Universal Robots PolyScope program: base_b.urp

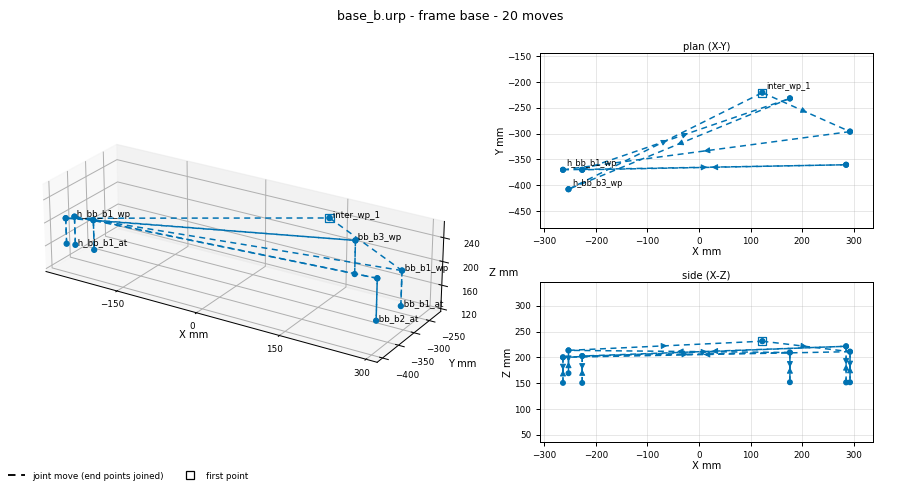
[picture p0: tool path of base_b.urp in frame base, 20 of 20 moves have a stored position in this frame; points joined in program order, loops and branches not executed]
Program base_b (installation=default directory=/programs/Session 1 createdIn=5.3.1.64192 lastSavedIn=5.3.1.64192 robotSerialNumber=20195300365)
Calibrated DH parameters: a=[-0.000093, -0.190649, -0.212673, 0.000091, -0.000205, 0]; d=[0.151591, 44.061648, -42.488068, -1.442789, 0.085322, 0.091911]; alpha=[1.570082, -0.003447, 0.007513, 1.572293, -1.571904, 0]; deltaTheta=[0, -0.672656, 0.728185, -0.055522, 0.000005, 0]
Robot Program (runOnlyOnce=true)
  URCap Gripper Activate (Robotiq_Grippers, Robotiq Inc.) dataModel(ResetAndActivateKey=false)
  URCap Gripper (Robotiq_Grippers, Robotiq Inc.) dataModel(position=50.0, force=100.0, speed=100.0, positionInDouble=50.0, forceInDouble=100.0, speedInDouble=100.0, slaveIds=[9], blocking=true)
  MoveJ speed 60 deg/s, acceleration 80 deg/s^2 (useActiveTCP=true) feature=Base
    Waypoint inter_wp_1: TCP in base x=122.78 y=-220.583 z=231.495 mm, rx=2.2968 ry=2.1205 rz=-0.0201 rad; joints [-29.631, -72.124, -124.848, -72.343, 89.412, -204.687] deg
  Folder Base_B
    MoveJ speed 60 deg/s, acceleration 80 deg/s^2 (useActiveTCP=true) feature=Base
      Waypoint bb_b1_wp: TCP in base x=292.658 y=-296.109 z=211.213 mm, rx=2.2199 ry=2.2113 rz=-0.0547 rad; joints [-26.688, -116.102, -82.488, -71.567, 88.238, -206.181] deg
      Waypoint bb_b1_at: TCP in base x=292.645 y=-296.127 z=151.887 mm, rx=2.2199 ry=2.2112 rz=-0.0548 rad; joints [-26.711, -122.1, -90.484, -57.573, 88.188, -206.122] deg
      URCap Gripper (Robotiq_Grippers, Robotiq Inc.) dataModel(position=100.0, force=100.0, speed=100.0, positionInDouble=100.0, forceInDouble=100.0, speedInDouble=100.0, slaveIds=[9], blocking=true)
      Waypoint bb_b1_wp: TCP in base x=292.658 y=-296.109 z=211.213 mm, rx=2.2199 ry=2.2113 rz=-0.0547 rad; joints [-26.688, -116.102, -82.488, -71.567, 88.238, -206.181] deg
      Waypoint h_bb_b1_wp: TCP in base x=-263.499 y=-370.068 z=200.329 mm, rx=-3.0828 ry=0.0524 rz=-0.0261 rad; joints [-108.781, -127.406, -65.833, -80.171, 90.182, -196.637] deg
      Waypoint h_bb_b1_at: TCP in base x=-263.484 y=-370.083 z=150.732 mm, rx=-3.0828 ry=0.0523 rz=-0.026 rad; joints [-108.797, -131.383, -72.897, -69.13, 90.158, -196.59] deg
      URCap Gripper (Robotiq_Grippers, Robotiq Inc.) dataModel(position=50.0, force=100.0, speed=100.0, positionInDouble=50.0, forceInDouble=100.0, speedInDouble=100.0, slaveIds=[9], blocking=true)
      Waypoint h_bb_b1_wp: TCP in base x=-263.499 y=-370.068 z=200.329 mm, rx=-3.0828 ry=0.0524 rz=-0.0261 rad; joints [-108.781, -127.406, -65.833, -80.171, 90.182, -196.637] deg
    MoveJ speed 60 deg/s, acceleration 80 deg/s^2 (useActiveTCP=true) feature=Base
      Waypoint bb_b2_wp: TCP in base x=285.029 y=-360.313 z=221.676 mm, rx=2.2402 ry=2.1488 rz=-0.0282 rad; joints [-34.898, -125.685, -65.053, -77.312, 88.836, -212.332] deg
      Waypoint bb_b2_at: TCP in base x=285.033 y=-360.322 z=151.608 mm, rx=2.2401 ry=2.1488 rz=-0.028 rad; joints [-34.925, -131.234, -75.256, -61.556, 88.801, -212.266] deg
      URCap Gripper (Robotiq_Grippers, Robotiq Inc.) dataModel(position=100.0, force=100.0, speed=100.0, positionInDouble=100.0, forceInDouble=100.0, speedInDouble=100.0, slaveIds=[9], blocking=true)
      Waypoint bb_b2_wp: TCP in base x=285.029 y=-360.313 z=221.676 mm, rx=2.2402 ry=2.1488 rz=-0.0282 rad; joints [-34.898, -125.685, -65.053, -77.312, 88.836, -212.332] deg
      Waypoint h_bb_b2_wp: TCP in base x=-226.231 y=-370.058 z=202.804 mm, rx=-3.101 ry=0.0514 rz=-0.0119 rad; joints [-103.98, -121.699, -75.13, -75.447, 90.191, -191.835] deg
      Waypoint h_bb_b2_at: TCP in base x=-226.246 y=-370.053 z=150.663 mm, rx=-3.101 ry=0.0514 rz=-0.0119 rad; joints [-104.001, -126.505, -82.189, -63.582, 90.158, -191.786] deg
      URCap Gripper (Robotiq_Grippers, Robotiq Inc.) dataModel(position=50.0, force=100.0, speed=100.0, positionInDouble=50.0, forceInDouble=100.0, speedInDouble=100.0, slaveIds=[9], blocking=true)
      Waypoint h_bb_b2_wp: TCP in base x=-226.231 y=-370.058 z=202.804 mm, rx=-3.101 ry=0.0514 rz=-0.0119 rad; joints [-103.98, -121.699, -75.13, -75.447, 90.191, -191.835] deg
    MoveJ speed 60 deg/s, acceleration 80 deg/s^2 (useActiveTCP=true) feature=Base
      Waypoint bb_b3_wp: TCP in base x=176.16 y=-231.769 z=209.637 mm, rx=-2.2431 ry=-2.1874 rz=-0.0349 rad; joints [-26.842, -86.447, -119.81, -63.708, 91.685, -204.985] deg
      Waypoint bb_b3_at: TCP in base x=176.163 y=-231.779 z=151.997 mm, rx=-2.2432 ry=-2.1874 rz=-0.0349 rad; joints [-26.868, -95.964, -129.106, -44.891, 91.583, -204.91] deg
      URCap Gripper (Robotiq_Grippers, Robotiq Inc.) dataModel(position=100.0, force=100.0, speed=100.0, positionInDouble=100.0, forceInDouble=100.0, speedInDouble=100.0, slaveIds=[9], blocking=true)
      Waypoint bb_b3_wp: TCP in base x=176.16 y=-231.769 z=209.637 mm, rx=-2.2431 ry=-2.1874 rz=-0.0349 rad; joints [-26.842, -86.447, -119.81, -63.708, 91.685, -204.985] deg
      Waypoint h_bb_b3_wp: TCP in base x=-252.791 y=-407.786 z=213.756 mm, rx=2.2404 ry=2.1812 rz=0.0538 rad; joints [-106.357, -133.377, -52.558, -85.313, 91.957, -284.711] deg
      Waypoint h_bb_b3_at: TCP in base x=-252.772 y=-407.793 z=169.415 mm, rx=2.2404 ry=2.1812 rz=0.0537 rad; joints [-106.375, -135.74, -60.423, -75.082, 91.946, -284.663] deg
      URCap Gripper (Robotiq_Grippers, Robotiq Inc.) dataModel(position=50.0, force=100.0, speed=100.0, positionInDouble=50.0, forceInDouble=100.0, speedInDouble=100.0, slaveIds=[9], blocking=true)
      Waypoint h_bb_b3_wp: TCP in base x=-252.791 y=-407.786 z=213.756 mm, rx=2.2404 ry=2.1812 rz=0.0538 rad; joints [-106.357, -133.377, -52.558, -85.313, 91.957, -284.711] deg
  MoveJ speed 60 deg/s, acceleration 80 deg/s^2 (useActiveTCP=true) feature=Base
    Waypoint inter_wp_1: TCP in base x=122.78 y=-220.583 z=231.495 mm, rx=2.2968 ry=2.1205 rz=-0.0201 rad; joints [-29.631, -72.124, -124.848, -72.343, 89.412, -204.687] deg
